FUNCTION_BLOCK FB_SaMElementNotAllowed EXTENDS FB_SaMElement
VAR
END_VAR

END_FUNCTION_BLOCK

(* stored: Version 1.1.0.1
   POU FB_SaMElementNotAllowed: Id {ae117149-e84b-087b-1b42-773e441658e5}, SpecialFunc None *)
